# EPICS autosave request: iocBoot/iocmcam/auto_settings.req
$(BL):$(DEV):mode
$(BL):$(DEV):resolution
$(BL):$(DEV):fps
